FUNCTION_BLOCK AnalogInput_Generic EXTENDS AnalogInput IMPLEMENTS I_AnalogChannel_Generic
VAR
	Status : REFERENCE TO ST_AnalogInputStatus_Generic;
END_VAR

PROPERTY DataValid : BOOL
GET
DataValid := NOT Status.WcState;
END_GET
END_PROPERTY

PROPERTY Error : BOOL
GET
Error := Status.Error;
END_GET
END_PROPERTY

(*FB_Init is always available implicitly and it is used primarily for initialization.
The return value is not evaluated. For a specific influence, you can also declare the
methods explicitly and provide additional code there with the standard initialization
code. You can evaluate the return value.*)
METHOD FB_Init : BOOL
VAR_INPUT
	(* TRUE: the retain variables are initialized (reset warm / reset cold)*)
	bInitRetains : BOOL;

	(* TRUE: the instance will be copied to the copy code afterward (online change)   *)
	bInCopyCode : BOOL;
	Name		: T_MaxString;
	Input		: REFERENCE TO INT;
	Status		: REFERENCE TO ST_AnalogInputStatus_Generic;
END_VAR
THIS^.Status REF= Status;
END_METHOD

PROPERTY Overrange : BOOL
GET
Overrange := Status.Overrange;
END_GET
END_PROPERTY

PROPERTY Underrange : BOOL
GET
Underrange := Status.Underrrange;
END_GET
END_PROPERTY

END_FUNCTION_BLOCK

(* stored: Version 1.1.0.1, ProductVersion 3.1.4026.18
   POU AnalogInput_Generic: Id {7006ea13-0319-435d-bd2c-84f4ad6c4b53}, SpecialFunc None
   Property DataValid: Id {85d1b353-1b29-425a-8738-e425d2e44b86}
   Get Get: Id {8579ea41-eea0-4d83-8545-db480a9f4fdd}
   Property Error: Id {bc28f45a-8845-44bb-972d-6e0ce157f873}
   Get Get: Id {dd4bbc4a-5d03-4f8c-9ddc-4eb35196ee7b}
   Method FB_Init: Id {84513803-f99a-4713-abd9-20afd4f4c4df}
   Property Overrange: Id {81485b52-bd22-41e7-8c93-567074bf9e15}
   Get Get: Id {47797d4a-c625-414b-addc-3b5d8b78adc0}
   Property Underrange: Id {45cca0c6-4763-4441-8500-1cf395e53001}
   Get Get: Id {f3a077e2-abe6-4d43-b57b-5487bbefb4f9} *)
